FUNCTION F_CreateDynTextEx : ST_Text
VAR_INPUT
	nNameId		: INT;		//example simatic hmi
	wsNameId	: WSTRING;	//standard name
	wsName		: WSTRING;	//standard name
END_VAR

F_CreateDynTextEx.nNameId := nNameId;
F_CreateDynTextEx.wsNameId := wsNameId;
F_CreateDynTextEx.wsName := wsName;

END_FUNCTION

(* stored: Version 1.1.0.1, ProductVersion 3.1.4024.12
   POU F_CreateDynTextEx: Id {c52bd20c-0ebc-4f65-b00e-7bb9df2b34fd}, SpecialFunc None *)
